Staubli VAL3: BitWord.pgx

public program BitWord(num x_nDecimal, string& x_sBinary[])
  local num l_ni
  local string l_sVal
begin
  //-----------------------------------------------------------------------
  //Header begin
  //Description of program
  //  This program turns a decimal number into a binary word.
  //  Receives decimal value and turns it into the corresponding
  //  binary word (16 Bits).
  //
  //Input parameters
  //  num x_nDecimal :
  //    role : decimal value to convert
  //
  //Output parameters
  //  string x_sBinary :
  //    role : binary value converted (16 Bits)
  //
  //Example
  //  BitWord(78,sBinaryValue)
  //
  //History
  //  Creation : 16-04-09 - t.Gra
  //Header end
  //-----------------------------------------------------------------------
  //take the full value
  x_nDecimal=roundDown(x_nDecimal)
  //Calcul loop
  do
    if (x_nDecimal%2)==0
      x_sBinary="0"+x_sBinary
    else
      x_sBinary="1"+x_sBinary
    endIf
    x_nDecimal=roundDown(x_nDecimal/2)
  until (x_nDecimal<1)
  l_sVal=x_sBinary
  //Add bit 0
  for l_ni=1 to (16-len(l_sVal))
    x_sBinary="0"+x_sBinary
  endFor
end
